// TwinCAT 3 PLC project Untitled1
// ProgramVersion: 3.1.4024.0
// libraries:
//   Tc2_Standard, * (Beckhoff Automation GmbH)
//   Tc2_System, * (Beckhoff Automation GmbH)
//   Tc3_Module, * (Beckhoff Automation GmbH)
//   Tc3_Vision, * (Beckhoff Automation GmbH)
// project tree:
//   / PlcTask.TcTTO
//   POUs/ AdaptiveThreshold.TcPOU, BlobDecect.TcPOU, MAIN.TcPOU
// real-time tasks:
//   TASK PlcTask: cycle T#100000us, priority 20, ADS port 350
//   TASK VnTask ImgAcq (FileSource1): cycle T#10ms, priority 5, ADS port 351
//   TASK JobTask_0: cycle default, priority 1
//   TASK JobTask_1: cycle default, priority 2
//   TASK JobTask_2: cycle default, priority 3
//   TASK JobTask_3: cycle default, priority 4

CONFIGURATION Untitled1
    RESOURCE PLC ON TwinCAT3
        TASK PlcTask(INTERVAL := T#100000us, PRIORITY := 20);
        PROGRAM MAIN WITH PlcTask : MAIN;
    END_RESOURCE
END_CONFIGURATION

// ---- POUs/MAIN.TcPOU
PROGRAM MAIN
VAR
	fbCamera			:	FB_VN_SimpleCameraControl;
	eState				:	ETcVnCameraState;	

	fbAdaptiveThreshold: AdaptiveThreshold();
	fbBlobDecect: BlobDecect();
END_VAR

//fbAdaptiveThreshold(fbCamera:=fbCamera,eState:=eState);
fbBlobDecect(fbCamera:=fbCamera,eState:=eState);

END_PROGRAM

// ---- POUs/AdaptiveThreshold.TcPOU
FUNCTION_BLOCK AdaptiveThreshold

VAR_INPUT
		// Camera
	fbCamera			:	REFERENCE TO FB_VN_SimpleCameraControl;
	eState				:	REFERENCE TO ETcVnCameraState;
END_VAR

VAR
	// Images
	ipImageIn			:	ITcVnImage;
	ipImageGrey		:	ITcVnImage;
	ipImageAdaptiveThreshold:	ITcVnImage;
	ipImageInDisp		:	ITcVnDisplayableImage;


		// Bilateral Filter
	ipImageFiltered		:	ITcVnImage;
	nBilateral_Diameter		:	DINT	:=	7;
	fBilateral_SigmaColor	:	LREAL	:=	20;
	fBilateral_SigmaSpace	:	LREAL	:=	100;
	
	
	ipImageAdaptiveThresholdDisp:	ITcVnDisplayableImage;
	
	// Contours
	ipContours		:	ITcVnContainer;		
	ipContour			:	ITcVnContainer;	
	ipIterator			:	ITcVnForwardIterator;
	ipIteratorFilteredList: ITcVnForwardIterator;
	ipContoursFiltered 		: ITcVnContainer;
	ipContourReference	:	ITcVnContainer;
	ipContourCheck		:	ITcVnContainer;
	ipContourPicked		:	ITcVnContainer;
	fBestDissimilarity	:	LREAL;
	fDissimilarity		:	LREAL;
	
	// Parameters Blob
	fThreshold			:	REAL := 170;
	fMinArea			:	REAL := 300;
	fMaxArea			:   LREAL :=1000;
	fMaxDissimilarity	:	LREAL := 0.01;
	eComparisonMethod	:	ETcVnContoursMatchComparisonMethod := TCVN_CMCM_CONTOURS_MATCH_I3;
	eThresholdType: ETcVnThresholdType;
	
	// Drawing
	aColorGreen			:	TcVnVector4_LREAL := [0, 175, 0];
	aColorBlue			:	TcVnVector4_LREAL := [0, 0, 255];
	aColorRed			:	TcVnVector4_LREAL := [255, 0, 0];
	aColorRes			:	TcVnVector4_LREAL;
	sContourNumberText				:	STRING(255);
	sTextReference		:	STRING(255) := 'Reference contour';
	sTextCheck			:	STRING(255) := 'Check dissimilarity';
	
		

		
	// Miscellaneous
	bDarkBackground		:	BOOL;
	nContours			:	ULINT;
	nCounter			:	UINT := 0;
	aPixelValue			:	TcVnVector4_LREAL;
	stBoundingRectangle	:	TcVnRectangle_UDINT;
	stParams			:	TcVnParamsBlobDetection;
	hr 					:	HRESULT;	



	
	aPosition: TcVnPoint2_DINT;
	aMaxValue: TcVnVector4_LREAL;

	
	//FindContoursExp
		eRetrievalMode: ETcVnContourRetrievalMode;
	eApproximationMethod: ETcVnContourApproximationMethod;
	aOffset: TcVnPoint;
	
	//Sorting list
	fArea: LREAL;
	
	// Watchdog
	hrWD 					:	HRESULT;
	tWDStop					:	DINT := 80000;	(* Stop time in us *)
	tRest 					:	DINT;
	nFunctionsMonitored		:	ULINT;
	nFractionProcessed 		:	UDINT;	
	tDuration 				:	DINT;
	

	Index: ULINT;
	ipSingleContour: INT;
	nContoursFiltered: ULINT;
	aCenter: TcVnPoint2_LREAL;
	fArea2: LREAL;
	reaknare: INT;
	
	
	//Create Structuring element for the Closing operation
ipStructuringElement: ITcVnImage;
eShape: ETcVnStructuringElementShape :=TCVN_SES_RECTANGLE;
	
	
	fAreaPicked: LREAL;
END_VAR



eState := fbCamera.GetState();

CASE eState OF

TCVN_CS_INITIAL, TCVN_CS_INITIALIZING, TCVN_CS_INITIALIZED, TCVN_CS_OPENING, TCVN_CS_OPENED, TCVN_CS_STARTACQUISITION:
	hr := fbCamera.StartAcquisition();

TCVN_CS_ACQUIRING:
	hr := fbCamera.GetCurrentImage(ipImageIn);	
	


	IF SUCCEEDED(hr) AND ipImageIn <> 0 THEN
		
		// Prepare result image
		hr := F_VN_ConvertColorSpace(ipImageIn, ipImageGrey, TCVN_CST_RGB_TO_GRAY, hr);
		//F_VN_MaxPixelValue(ipImageIn,aMaxValue,aPosition,hr);
		//F_VN_MinPixelValue(ipImageIn,aMaxValue,aPosition,hr);
		//hr:=F_VN_NormalizeImage(ipImageIn,ipImageIn,hr);




		
//Start watchdog to limit the time allowed for the functions below. 
		hrWD := F_VN_StartRelWatchdog(tWDStop, hr);
		
		
//		//Filter image smooth.
//			hr := F_VN_GaussianFilterExp(
//			ipSrcImage      :=  ipImageIn,
//			ipDestImage     :=  ipImageFiltered,
//			nFilterWidth    :=  3,
//			nFilterHeight   :=  3,
//			fSigmaX         :=  5,
//			fSigmaY         :=  5,
//			eBorderType     :=  TCVN_BIM_DEFAULT,
//			hrPrev          :=  hr
//			);
			
//			hr := F_VN_BilateralFilter(
//						ipSrcImage      :=  ipImageIn,
//						ipDestImage     :=  ipImageFiltered,
//						nDiameter       :=  nBilateral_Diameter,//dDiameter set to 0 for automatic calculation depending on fSigmaSpace
//						fSigmaColor     :=  fBilateral_SigmaColor,
//						fSigmaSpace     :=  fBilateral_SigmaSpace,
//						hrPrev          :=  hr);

			//	hr := F_VN_CopyIntoDisplayableImage(ipImageFiltered, ipImageFilteredDisp, hr);			
						
	
	hr := F_VN_AdaptiveThresholdExp(
    ipSrcImage      :=  ipImageGrey,
    ipDestImage     :=  ipImageAdaptiveThreshold, 
    fMaxValue       :=  255, // max value of 8-bit image: (2^8)-1=255
    eAdaptiveMethod :=  TCVN_ATM_MEAN,
    eThresholdType  :=  TCVN_TT_BINARY_INV, //TCVN_TT_BINARY_INV,
    nBlockSize      :=  5,
    fConstant       :=  10,
    hrPrev          :=  hr
);

		hr := F_VN_CopyIntoDisplayableImage(ipImageAdaptiveThreshold, ipImageAdaptiveThresholdDisp, hr);


		hr:= F_VN_CreateStructuringElement(ipStructuringElement,eShape, 3, 3, hr);	
	
		//	hr:= F_VN_MorphologicalOperator(ipImageAdaptiveThreshold, ipImageAdaptiveThreshold, TCVN_MO_EROSION,ipStructuringElement, hr);
//			hr:= F_VN_MorphologicalOperator(ipImageAdaptiveThreshold, ipImageAdaptiveThreshold, TCVN_MO_CLOSING,ipStructuringElement, hr);
		//	hr:= F_VN_MorphologicalOperator(ipImageAdaptiveThreshold, ipImageAdaptiveThreshold, TCVN_MO_DILATION,ipStructuringElement, hr);



		hr:=F_VN_FindContoursExp(ipImageAdaptiveThreshold,ipContours,eRetrievalMode,eApproximationMethod,aOffset,hr);

		hr := F_VN_GetNumberOfElements(ipContours, nContours, hr);

		
		
//		//Blob detection
//		stParams.bFilterByArea:= TRUE;
//		stParams.fMinArea:=fMinArea;
//		stParams.fMaxArea:=fMaxArea;
//		stParams.bFilterByCircularity:=FALSE;
//		//stParams.fMaxCircularity:=0.9;
//		stParams.fMinThreshold:=150;
		stParams.eThresholdType:= eThresholdType;
		
//		hr := F_VN_DetectBlobs(ipImageIn, ipContours, stParams, hr);


		
	//Stop watchdog to limit the time allowed for the functions above. 
hrWD := F_VN_StopWatchdog(hrWD, nFunctionsMonitored => nFunctionsMonitored, nFractionProcessed => nFractionProcessed, tRest => tRest);


		//Testkod för att filtrera ut bara vissa konturer 
			
			//Skapa ny filtrerad lista av konturer
			hr:= F_VN_CreateContainer(ipContoursFiltered, ContainerType_Vector_Vector_TcVnPoint2_DINT,0, hr);  
			hr:= F_VN_ReserveContainerMemory(ipContoursFiltered, 100, hr);  //Only for performance reasons		
		
			hr := F_VN_GetForwardIterator(ipContours, ipIterator, hr);
			hr := F_VN_GetForwardIterator(ipContoursFiltered, ipIteratorFilteredList, hr);


			
					
			//Loop through every contour and filter it into a new list
		WHILE SUCCEEDED(hr) AND_THEN ipIterator.CheckIfEnd() <> S_OK DO

			hr:= F_VN_GetContainer(ipIterator, ipContour, hr);
					hr:= F_VN_ContourArea(ipContour, fArea, hr);
					
				IF fArea > 300  AND fArea < 1400 THEN
								hr:=F_VN_InsertIntoContainer_ITcVnContainer(ipContour,ipContoursFiltered,Index, hr);

								IF index= 2 THEN
										hr:= F_VN_ContourArea(ipContour, fArea2, hr);
								END_IF

								Index:=Index+1;		
								
								hr:= F_VN_ContourCenterOfMass(ipContour, aCenter, hr);
								sContourNumberText:= ULINT_TO_STRING(index);						
			hr:= F_VN_PutText(sContourNumberText, ipImageIn, LREAL_TO_UDINT(aCenter[0])+10,LREAL_TO_UDINT(aCenter[1]), ETcVnFontType.TCVN_FT_HERSHEY_PLAIN, 2, aColorGreen, hr);					
				END_IF
		
			hr:= F_VN_IncrementIterator(ipIterator, hr);
			
		END_WHILE

				hr := F_VN_GetNumberOfElements(ipContoursFiltered, nContoursFiltered, hr);
	
			//Get information about a specific contour			
				IF nContoursFiltered > 0 THEN
						hr := F_VN_GetAt_ITcVnContainer(ipContours, ipContourPicked, 39, hr);
						hr:= F_VN_ContourArea(ipContourPicked, fAreaPicked, hr);
				END_IF
			



		
					// Select one of the found contours as reference for matching
			hr := F_VN_GetAt_ITcVnContainer(ipContours, ipContourReference, nCounter MOD nContours, hr);

			// Draw selected contour and text
						reaknare:=(reaknare +1)MOD 1000 ;
						sTextReference:= INT_TO_STRING(reaknare);
			hr := F_VN_PutTextExp(sTextReference, ipImageIn, 50, 150, TCVN_FT_HERSHEY_SIMPLEX, 2.3, aColorBlue, 3, TCVN_LT_8_CONNECTED, FALSE, hr);
			hr := F_VN_DrawContours(ipContourReference, -1, ipImageIn, aColorBlue, 5, hr);

		Index:=0;
		
		hr:= F_VN_DrawContours(ipContoursFiltered, -1, ipImageIn, aColorRed, 2, hr);
		//		hr := F_VN_DrawContours(ipContours, -1, ipImageIn, aColorGreen, 1, hr);
			
//		
//				hr :=	F_VN_MatchContours(ipContour ,ipReference_Triangle, TCVN_CMCM_CONTOURS_MATCH_I1, fDissimilarity, hr);

					
//				END_IF
//			ELSE
//				sContourNumberText:= 'Red';		
//			END_IF
//			hr:= F_VN_ContourCenterOfMass(ipContour, aCenter, hr);
//			hr1:= F_VN_PutText(sContourNumberText, ipImageResult, LREAL_TO_UDINT(aCenter[0])+100,LREAL_TO_UDINT(aCenter[1]), ETcVnFontType.TCVN_FT_HERSHEY_PLAIN, 2, aColor_red, hr);
				
		
		



			
			nCounter := nCounter + 1;
		
		ELSE
			
//			fBestDissimilarity := 10E300;
			
//			// Iterate through all found contours

//			WHILE hr = S_OK AND_THEN ipIterator.CheckIfEnd() <> S_OK DO
//				hr := F_VN_GetContainer(ipIterator, ipContourCheck, hr);
//				hr := F_VN_IncrementIterator(ipIterator, hr);
				
//				// Match the current contour with the selected reference contour
//				hr := F_VN_MatchContours(ipContourReference, ipContourCheck, eComparisonMethod, fDissimilarity, hr);
				
//				// Save best result
//				IF fBestDissimilarity > fDissimilarity THEN
//					fBestDissimilarity := fDissimilarity;
//				END_IF
				
//				// Choose action depending on the dissimilarity of both contours
//				IF SUCCEEDED(hr) AND_THEN fDissimilarity < fMaxDissimilarity THEN
//					aColorRes := aColorGreen;
//				ELSE
//					aColorRes := aColorRed;
//				END_IF
				
//				// Draw matching results
//				sContourNumberText := REAL_TO_STRING(LREAL_TO_REAL(fDissimilarity));
//				hr := F_VN_UprightBoundingRectangle(ipContourCheck, stBoundingRectangle, hr);
//				hr := F_VN_DrawContours(ipContourCheck, -1, ipImageIn, aColorRes, 5, hr);
//				hr := F_VN_PutTextExp(sContourNumberText, ipImageIn, LREAL_TO_UDINT(stBoundingRectangle.nX + 30), LREAL_TO_UDINT(stBoundingRectangle.nY + (stBoundingRectangle.nHeight / 2)), TCVN_FT_HERSHEY_SIMPLEX, 0.8, aColorRes, 2, TCVN_LT_8_CONNECTED, FALSE, hr);

//			END_WHILE
			
//			// Draw text
//			hr := F_VN_PutTextExp(sTextCheck, ipImageIn, 50, 50, TCVN_FT_HERSHEY_SIMPLEX, 1.3, aColorGreen, 2, TCVN_LT_8_CONNECTED, FALSE, hr);
//			sContourNumberText := CONCAT('Best match: ', REAL_TO_STRING(LREAL_TO_REAL(fBestDissimilarity)));
//			hr := F_VN_PutTextExp(sContourNumberText, ipImageIn, 50, 100, TCVN_FT_HERSHEY_SIMPLEX, 1.3, aColorGreen, 2, TCVN_LT_8_CONNECTED, FALSE, hr);
			
		END_IF

		
		hr := F_VN_CopyIntoDisplayableImage(ipImageIn, ipImageInDisp, hr);



	
TCVN_CS_ERROR:
	hr := fbCamera.Reset();	

END_CASE

END_FUNCTION_BLOCK

// ---- POUs/BlobDecect.TcPOU
FUNCTION_BLOCK BlobDecect
VAR_INPUT
			// Camera
	fbCamera			:	REFERENCE TO FB_VN_SimpleCameraControl;
	eState				:	REFERENCE TO ETcVnCameraState;
END_VAR

VAR
		hr 					:	HRESULT;	

	//Images		
	ipImageIn				:	ITcVnImage;
	ipImageGrey				:	ITcVnImage;
	ipImageInDisp			:	ITcVnDisplayableImage;
	
	// Watchdog
	hrWD 					:	HRESULT;
	tWDStop					:	DINT := 80000;	(* Stop time in us *)
	tRest 					:	DINT;
	nFunctionsMonitored		:	ULINT;
	nFractionProcessed 		:	UDINT;	
	tDuration 				:	DINT;
	
			// Bilateral Filter
	ipImageFiltered		:	ITcVnImage;
	nBilateral_Diameter		:	DINT	:=	7;
	fBilateral_SigmaColor	:	LREAL	:=	20;
	fBilateral_SigmaSpace	:	LREAL	:=	100;
	
	
	
	
		// Contours
	ipContours		:	ITcVnContainer;	
	ipContour			:	ITcVnContainer;	
	ipIterator			:	ITcVnForwardIterator;
	ipContoursFiltered 		: ITcVnContainer;
	ipIteratorFilteredList: ITcVnForwardIterator;
	nContours			:	ULINT;
	nContoursFiltered: ULINT;
	ipContourPicked		:	ITcVnContainer;
	fAreaPicked: LREAL;
	nContourMaster: ULINT:= 2;
	
		// Parameters Blob
	stParams			:	TcVnParamsBlobDetection;	
	eThresholdType: ETcVnThresholdType;
	fThreshold			:	REAL := 170;
	fMinArea			:	REAL := 300;
	fMaxArea			:   LREAL :=1000;
	fMaxDissimilarity	:	LREAL := 0.01;
	eComparisonMethod	:	ETcVnContoursMatchComparisonMethod := TCVN_CMCM_CONTOURS_MATCH_I3;

	//Filtering Contours list
	fArea: LREAL;
	fCircularity: LREAL;
	fCircularityPicked: LREAL;
	Index: ULINT;
	aCenter: TcVnPoint2_LREAL;
	sContourNumberText: STRING;	
	stRectanglePicked: TcVnRotatedRectangle;
	RectangleDataForPicking: ARRAY [0..500] OF 	TcVnRotatedRectangle;
	// Drawing
	aColorGreen			:	TcVnVector4_LREAL := [0, 175, 0];
	aColorBlue			:	TcVnVector4_LREAL := [0, 0, 255];
	aColorRed			:	TcVnVector4_LREAL := [255, 0, 0];
	
	//Categorize products
	iNumberOfProducts: DINT;
	iCurrentProduct: ULINT;
	CurrentArea: REAL;
	nTolerance: REAL := 100;
	nAreaRectanglePicked: REAL;
END_VAR

eState := fbCamera.GetState();

CASE eState OF

TCVN_CS_INITIAL, TCVN_CS_INITIALIZING, TCVN_CS_INITIALIZED, TCVN_CS_OPENING, TCVN_CS_OPENED, TCVN_CS_STARTACQUISITION:
	hr := fbCamera.StartAcquisition();

TCVN_CS_ACQUIRING:
	hr := fbCamera.GetCurrentImage(ipImageIn);	
	


	IF SUCCEEDED(hr) AND ipImageIn <> 0 THEN
		
		// Prepare result image
		hr := F_VN_ConvertColorSpace(ipImageIn, ipImageGrey, TCVN_CST_RGB_TO_GRAY, hr);
		//F_VN_MaxPixelValue(ipImageIn,aMaxValue,aPosition,hr);
		//F_VN_MinPixelValue(ipImageIn,aMaxValue,aPosition,hr);
		//hr:=F_VN_NormalizeImage(ipImageIn,ipImageIn,hr);




		
//Start watchdog to limit the time allowed for the functions below. 
		hrWD := F_VN_StartRelWatchdog(tWDStop, hr);
		
		
//		//Filter image smooth.
//			hr := F_VN_GaussianFilterExp(
//			ipSrcImage      :=  ipImageIn,
//			ipDestImage     :=  ipImageFiltered,
//			nFilterWidth    :=  3,
//			nFilterHeight   :=  3,
//			fSigmaX         :=  5,
//			fSigmaY         :=  5,
//			eBorderType     :=  TCVN_BIM_DEFAULT,
//			hrPrev          :=  hr
//			);
			
//			hr := F_VN_BilateralFilter(
//						ipSrcImage      :=  ipImageIn,
//						ipDestImage     :=  ipImageFiltered,
//						nDiameter       :=  nBilateral_Diameter,//dDiameter set to 0 for automatic calculation depending on fSigmaSpace
//						fSigmaColor     :=  fBilateral_SigmaColor,
//						fSigmaSpace     :=  fBilateral_SigmaSpace,
//						hrPrev          :=  hr);

			//	hr := F_VN_CopyIntoDisplayableImage(ipImageFiltered, ipImageFilteredDisp, hr);			
			
			
		//Blob detection
		stParams.bFilterByArea:= TRUE;
		stParams.fMinArea:=fMinArea;
		stParams.fMaxArea:=fMaxArea;
//		stParams.bFilterByCircularity:=FALSE;
//		stParams.fMinCircularity:=0.15;
		stParams.fMinThreshold:=130;  //150 start value
		stParams.eThresholdType:= eThresholdType;
		
		hr := F_VN_DetectBlobs(ipImageIn, ipContours, stParams, hr);
				hr := F_VN_GetNumberOfElements(ipContours, nContours, hr);

//		hr:= F_VN_DrawContours(ipContours, -1, ipImageIn, aColorBlue, 2, hr);


			
	//Stop watchdog to limit the time allowed for the functions above. 
hrWD := F_VN_StopWatchdog(hrWD, nFunctionsMonitored => nFunctionsMonitored, nFractionProcessed => nFractionProcessed, tRest => tRest);


			//Skapa ny filtrerad lista av konturer
			hr:= F_VN_CreateContainer(ipContoursFiltered, ContainerType_Vector_Vector_TcVnPoint2_DINT,0, hr);  
			hr:= F_VN_ReserveContainerMemory(ipContoursFiltered, 100, hr);  //Only for performance reasons
			hr := F_VN_GetForwardIterator(ipContours, ipIterator, hr);
			hr := F_VN_GetForwardIterator(ipContoursFiltered, ipIteratorFilteredList, hr);

			//Loop through every contour and filter it into a new list
			Index:=0;
			WHILE SUCCEEDED(hr) AND_THEN ipIterator.CheckIfEnd() <> S_OK DO
				
				//Check area and circularity on current contour 
				hr:= F_VN_GetContainer(ipIterator, ipContour, hr);
						hr:= F_VN_ContourArea(ipContour, fArea, hr);
						hr:= F_VN_ContourCircularity(ipContour, fCircularity, hr);

					//Check if Contour meets area and circularity measures	
					IF fArea > 400  AND fArea < 1500 AND fCircularity > 0.15 THEN
									hr:=F_VN_InsertIntoContainer_ITcVnContainer(ipContour,ipContoursFiltered,Index, hr);					
									hr:= F_VN_ContourCenterOfMass(ipContour, aCenter, hr);
									sContourNumberText:= ULINT_TO_STRING(index);						
				hr:= F_VN_PutText(sContourNumberText, ipImageIn, LREAL_TO_UDINT(aCenter[0])+10,LREAL_TO_UDINT(aCenter[1]), ETcVnFontType.TCVN_FT_HERSHEY_PLAIN, 2, aColorGreen, hr);					
				F_VN_EnclosingRectangle(ipContour,RectangleDataForPicking[index], hr);
//				hr:= F_VN_DrawRotatedRectangle(RectangleDataForPicking[index],ipImageIn, aColorGreen,2,hr);
									Index:=Index+1;						
					END_IF
			
				hr:= F_VN_IncrementIterator(ipIterator, hr);
				
			END_WHILE

//					hr:= F_VN_DrawContours(ipContoursFiltered, -1, ipImageIn, aColorRed, 2, hr);
					
				//Get specific contour	- and pick as master for matching
				IF nContoursFiltered > nContourMaster  THEN				
						hr := F_VN_GetAt_ITcVnContainer(ipContoursFiltered, ipContourPicked, nContourMaster, hr);
						hr:=  F_VN_EnclosingRectangle(ipContourPicked,stRectanglePicked, hr);
						//hr:= F_VN_DrawContours(ipContoursFiltered,ULINT_TO_DINT(nContourMaster),ipImageIn,aColorGreen,2,hr);
						hr:= F_VN_ContourCircularity(ipContourPicked, fCircularityPicked, hr);
						hr:= F_VN_ContourArea(ipContourPicked, fAreaPicked, hr);
						nAreaRectanglePicked:= stRectanglePicked.stSize.fHeight*stRectanglePicked.stSize.fWidth;
						//Draw selected master contour
						hr:= F_VN_DrawRotatedRectangle(stRectanglePicked,ipImageIn, aColorBlue,3,hr);
						
				END_IF			
							hr := F_VN_GetNumberOfElements(ipContoursFiltered, nContoursFiltered, hr);


				//Categorize products
				FOR iCurrentProduct:= 0 TO nContoursFiltered DO
					CurrentArea:=RectangleDataForPicking[iCurrentProduct].stSize.fHeight * RectangleDataForPicking[iCurrentProduct].stSize.fWidth;
					IF CurrentArea-nTolerance < nAreaRectanglePicked AND CurrentArea+nTolerance > nAreaRectanglePicked THEN
						hr:= F_VN_DrawRotatedRectangle(RectangleDataForPicking[iCurrentProduct],ipImageIn, aColorGreen,3,hr);
					ELSE
						hr:= F_VN_DrawRotatedRectangle(RectangleDataForPicking[iCurrentProduct],ipImageIn, aColorRed,3,hr);

					END_IF
				END_FOR
				

		END_IF

		
		hr := F_VN_CopyIntoDisplayableImage(ipImageIn, ipImageInDisp, hr);



	
TCVN_CS_ERROR:
	hr := fbCamera.Reset();	

END_CASE

END_FUNCTION_BLOCK
